{attribute 'linkalways'} 
{attribute 'no_explicit_call' := 'This FB is a CLASS and must be accessed using methods or properties'}
{attribute 'enable_dynamic_creation'}
FUNCTION_BLOCK FINAL NE_BYTE EXTENDS Node
VAR
	in1 : _BYTE(0);
	in2 : _BYTE(0);
	out : _BOOL(FALSE);
END_VAR

METHOD PUBLIC Clone : I_Node
VAR
	pNode : POINTER TO NE_BYTE;
END_VAR
pNode := __NEW(NE_BYTE);
Clone := pNode^;
END_METHOD

METHOD FB_init : BOOL
VAR_INPUT
	bInitRetains : BOOL; // if TRUE, the retain variables are initialized (warm start / cold start)
	bInCopyCode : BOOL;  // if TRUE, the instance afterwards gets moved into the copy code (online change)
END_VAR
AddInput('in1',THIS^.in1);
AddInput('in2',THIS^.in2);
AddOutput('out', THIS^.out);
END_METHOD

METHOD PROTECTED OnExecute
VAR
END_VAR
out.Value := in1.Value <> in2.Value;
END_METHOD

END_FUNCTION_BLOCK

(* stored: Version 1.1.0.1, ProductVersion 3.1.4024.15
   POU NE_BYTE: Id {25503de4-dd8e-4091-8b2b-7576c50a9098}, SpecialFunc None
   Folder Constructor: Id {4a0249e8-b2ea-46cb-925b-e55d22b700cd}
   Method Clone: Id {57843909-d1f9-4cf7-93d8-67da34ce66bd}
   Method FB_init: Id {15573b59-e24f-4482-ad03-119c50d59ccb}
   Method OnExecute: Id {e7c39610-d3f8-4de7-929b-2f274b90629f} *)
